// Struckig
// Copyright (C) 2022 Stefan Besler

// This program is free software: you can redistribute it and/or modify
// it under the terms of the GNU General Public License as published by
// the Free Software Foundation, either version 3 of the License, or
// (at your option) any later version.

// This program is distributed in the hope that it will be useful,
// but WITHOUT ANY WARRANTY; without even the implied warranty of
// MERCHANTABILITY or FITNESS FOR A PARTICULAR PURPOSE.  See the
// GNU General Public License for more details.
//
// You should have received a copy of the GNU General Public License
// along with THIS PROGRAM.  IF NOT, see <http://www.gnu.org/licenses/>.
{attribute 'qualified_only'}
/// Error codes reported by the trajectory generator.
/// Returned by [ErrorCode](xref:Struckig.IOtg#ErrorCode) and explained by
/// [ErrorMessage](xref:Struckig.IOtg#ErrorMessage).
TYPE TrajectoryErrorCode :
(
  Undefined := 0, //< No error.
  InvalidInput, //< Error in the input parameter
  SynchronizationFailed, //< No valid synchronized profile was found.
  CalculateStep1Failed, //< Profile search in step 1 failed.
  ZeroLimitsConflict, //< Conflicting zero limits prevent profile generation.
  ZeroLimitsConflictInSynchronization //< Zero-limit conflict during multi-DoF synchronization.
);
END_TYPE

(* stored: Version 1.1.0.1
   DUT TrajectoryErrorCode: Id {b6f9027e-b647-46b0-a8f4-fdacb3d850bf} *)
